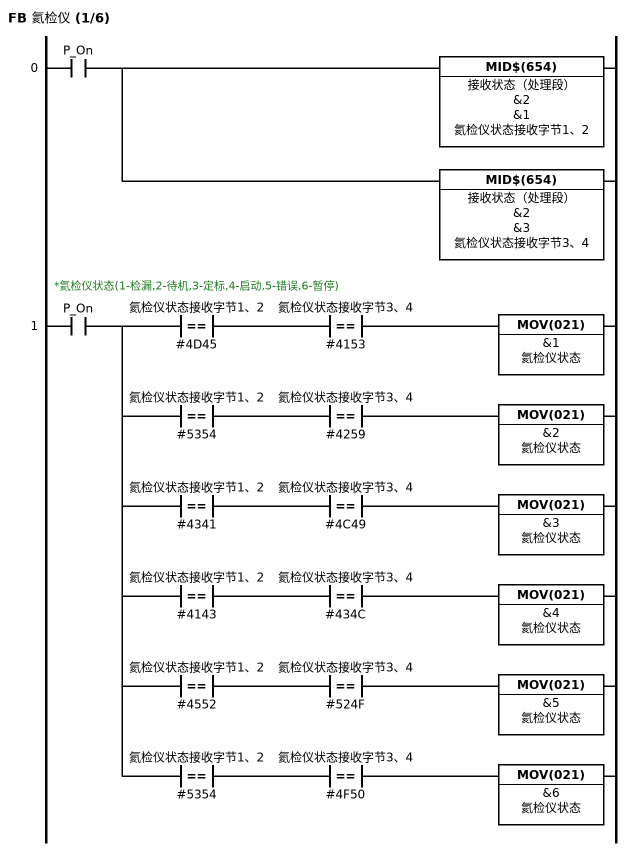
; rung 0
LD P_On
MID$(654) 接收状态（处理段） &2 &1 氦检仪状态接收字节1、2
MID$(654) 接收状态（处理段） &2 &3 氦检仪状态接收字节3、4
; rung 1: *氦检仪状态(1-检漏,2-待机,3-定标,4-启动,5-错误,6-暂停)
LD P_On
OUT TR0
AND=(300) 氦检仪状态接收字节1、2 #4D45
AND=(300) 氦检仪状态接收字节3、4 #4153
MOV(021) &1 氦检仪状态
LD TR0
AND=(300) 氦检仪状态接收字节1、2 #5354
AND=(300) 氦检仪状态接收字节3、4 #4259
MOV(021) &2 氦检仪状态
LD TR0
AND=(300) 氦检仪状态接收字节1、2 #4341
AND=(300) 氦检仪状态接收字节3、4 #4C49
MOV(021) &3 氦检仪状态
LD TR0
AND=(300) 氦检仪状态接收字节1、2 #4143
AND=(300) 氦检仪状态接收字节3、4 #434C
MOV(021) &4 氦检仪状态
LD TR0
AND=(300) 氦检仪状态接收字节1、2 #4552
AND=(300) 氦检仪状态接收字节3、4 #524F
MOV(021) &5 氦检仪状态
LD TR0
AND=(300) 氦检仪状态接收字节1、2 #5354
AND=(300) 氦检仪状态接收字节3、4 #4F50
MOV(021) &6 氦检仪状态

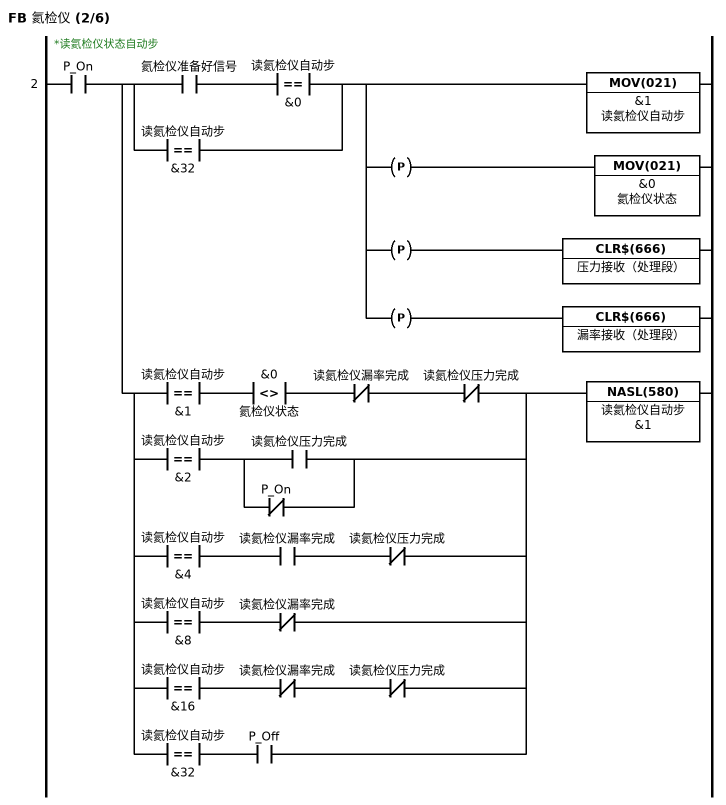
; rung 2: *读氦检仪状态自动步
LD P_On
OUT TR0
LD 氦检仪准备好信号
AND=(300) 读氦检仪自动步 &0
OR=(300) 读氦检仪自动步 &32
ANDLD
OUT TR1
MOV(021) &1 读氦检仪自动步
UP(521)
MOV(021) &0 氦检仪状态
LD TR1
UP(521)
CLR$(666) 压力接收（处理段）
LD TR1
UP(521)
CLR$(666) 漏率接收（处理段）
LD TR0
LD=(300) 读氦检仪自动步 &1
AND<>(305) &0 氦检仪状态
ANDNOT 读氦检仪漏率完成
ANDNOT 读氦检仪压力完成
LD=(300) 读氦检仪自动步 &2
LD 读氦检仪压力完成
ORNOT P_On
ANDLD
ORLD
LD=(300) 读氦检仪自动步 &4
AND 读氦检仪漏率完成
ANDNOT 读氦检仪压力完成
ORLD
LD=(300) 读氦检仪自动步 &8
ANDNOT 读氦检仪漏率完成
ORLD
LD=(300) 读氦检仪自动步 &16
ANDNOT 读氦检仪漏率完成
ANDNOT 读氦检仪压力完成
ORLD
LD=(300) 读氦检仪自动步 &32
AND P_Off
ORLD
ANDLD
NASL(580) 读氦检仪自动步 &1

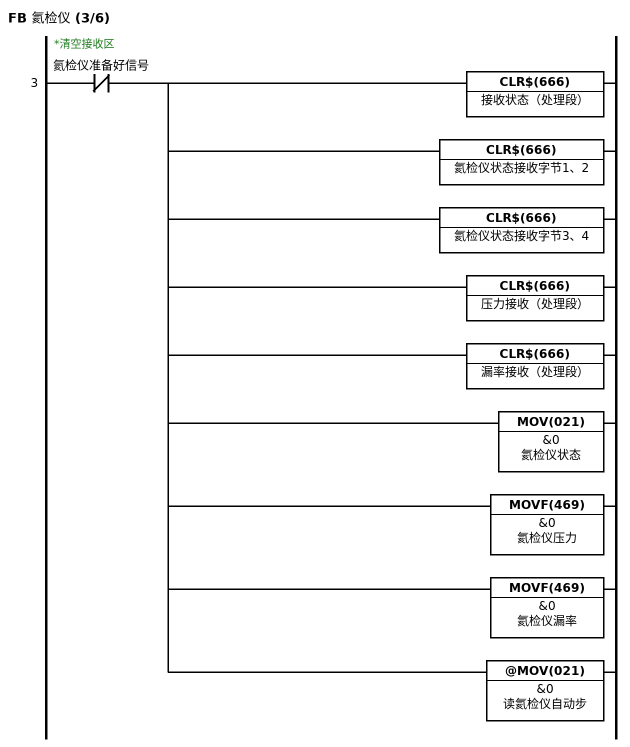
; rung 3: *清空接收区
LDNOT 氦检仪准备好信号
CLR$(666) 接收状态（处理段）
CLR$(666) 氦检仪状态接收字节1、2
CLR$(666) 氦检仪状态接收字节3、4
CLR$(666) 压力接收（处理段）
CLR$(666) 漏率接收（处理段）
MOV(021) &0 氦检仪状态
MOVF(469) &0 氦检仪压力
MOVF(469) &0 氦检仪漏率
@MOV(021) &0 读氦检仪自动步

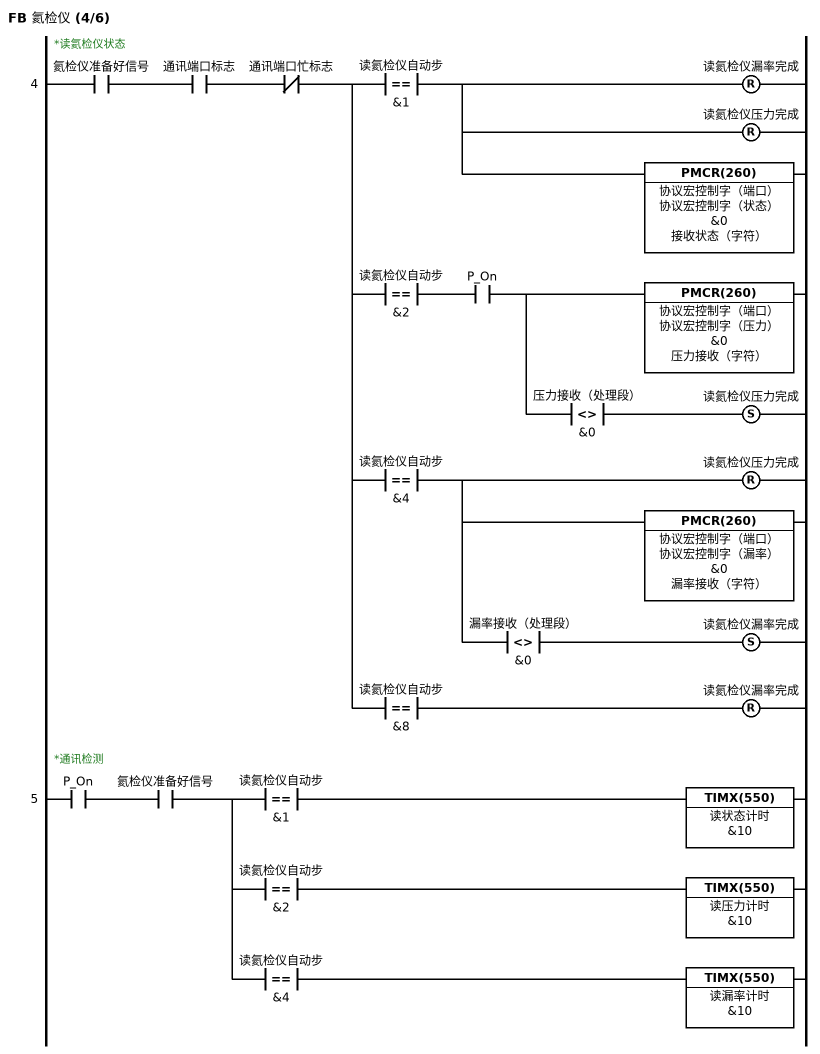
; rung 4: *读氦检仪状态
LD 氦检仪准备好信号
AND 通讯端口标志
ANDNOT 通讯端口忙标志
OUT TR0
AND=(300) 读氦检仪自动步 &1
RSET 读氦检仪漏率完成
RSET 读氦检仪压力完成
PMCR(260) 协议宏控制字（端口） 协议宏控制字（状态） &0 接收状态（字符）
LD TR0
AND=(300) 读氦检仪自动步 &2
AND P_On
PMCR(260) 协议宏控制字（端口） 协议宏控制字（压力） &0 压力接收（字符）
AND<>(305) 压力接收（处理段） &0
SET 读氦检仪压力完成
LD TR0
AND=(300) 读氦检仪自动步 &4
RSET 读氦检仪压力完成
PMCR(260) 协议宏控制字（端口） 协议宏控制字（漏率） &0 漏率接收（字符）
AND<>(305) 漏率接收（处理段） &0
SET 读氦检仪漏率完成
LD TR0
AND=(300) 读氦检仪自动步 &8
RSET 读氦检仪漏率完成
; rung 5: *通讯检测
LD P_On
AND 氦检仪准备好信号
OUT TR0
AND=(300) 读氦检仪自动步 &1
TIMX(550) 读状态计时 &10
LD TR0
AND=(300) 读氦检仪自动步 &2
TIMX(550) 读压力计时 &10
LD TR0
AND=(300) 读氦检仪自动步 &4
TIMX(550) 读漏率计时 &10

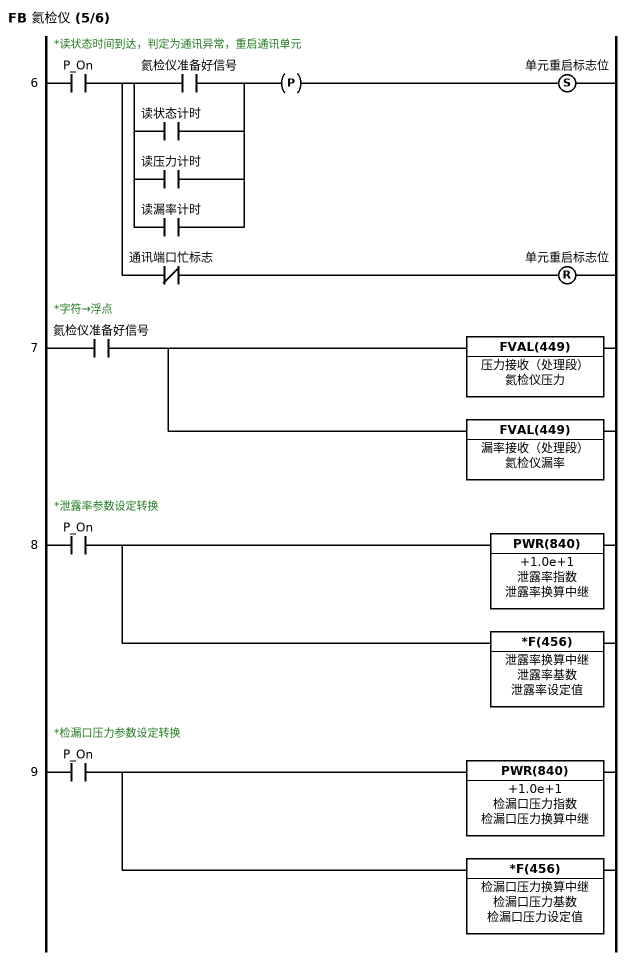
; rung 6: *读状态时间到达，判定为通讯异常，重启通讯单元
LD P_On
OUT TR0
LD 氦检仪准备好信号
OR 读状态计时
OR 读压力计时
OR 读漏率计时
ANDLD
UP(521)
SET 单元重启标志位
LD TR0
ANDNOT 通讯端口忙标志
RSET 单元重启标志位
; rung 7: *字符→浮点
LD 氦检仪准备好信号
FVAL(449) 压力接收（处理段） 氦检仪压力
FVAL(449) 漏率接收（处理段） 氦检仪漏率
; rung 8: *泄露率参数设定转换
LD P_On
PWR(840) +1.0e+1 泄露率指数 泄露率换算中继
*F(456) 泄露率换算中继 泄露率基数 泄露率设定值
; rung 9: *检漏口压力参数设定转换
LD P_On
PWR(840) +1.0e+1 检漏口压力指数 检漏口压力换算中继
*F(456) 检漏口压力换算中继 检漏口压力基数 检漏口压力设定值

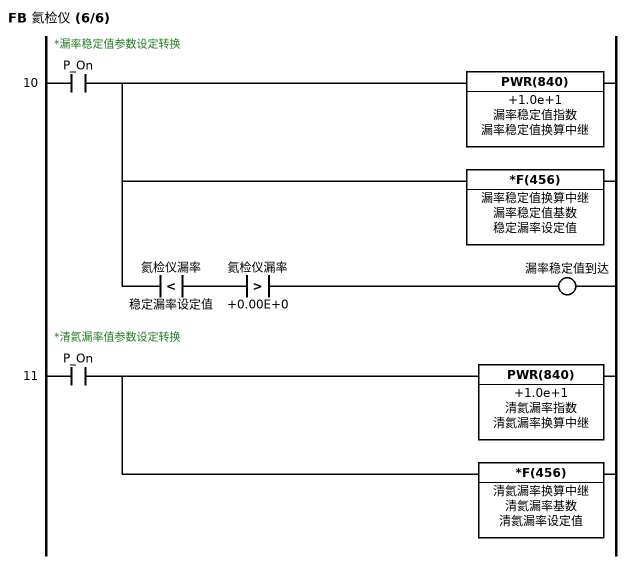
; rung 10: *漏率稳定值参数设定转换
LD P_On
PWR(840) +1.0e+1 漏率稳定值指数 漏率稳定值换算中继
*F(456) 漏率稳定值换算中继 漏率稳定值基数 稳定漏率设定值
AND<F(331) 氦检仪漏率 稳定漏率设定值
AND>F(333) 氦检仪漏率 +0.00E+0
OUT 漏率稳定值到达
; rung 11: *清氦漏率值参数设定转换
LD P_On
PWR(840) +1.0e+1 清氦漏率指数 清氦漏率换算中继
*F(456) 清氦漏率换算中继 清氦漏率基数 清氦漏率设定值

## Function block 腔体自检
VAR_INPUT
  紧急停止 : BOOL;
  真空泵启动信号 : BOOL;
  实时真空值 : REAL;
  自检抽真空设定阀值 : REAL;
  自检破真空设定阀值 : REAL;
  自检抽真空设定时间 : UINT;
  自检保压前设定时间 : UINT;
  自检保压设定时间 : UINT;
  自检泄漏量上限 : REAL;
  腔体顶升气缸上升到位信号 : BOOL;
  腔体顶升气缸下降到位信号 : BOOL;
  平移气缸出料位信号 : BOOL;
  平移气缸氦检位信号 : BOOL;
  抽真空阀状态 : BOOL;
  破真空阀状态 : BOOL;
  抽气阀可打开 : BOOL;
  自检停止（SW） : BOOL;
  自检启动（SW） : BOOL;
  工站初始化 : BOOL;
  腔体在初始位 : BOOL;
END_VAR
VAR_OUTPUT
  功能块运行中 : BOOL;
  自检保压前真空值（PV） : REAL;
  自检保压后真空值（PV） : REAL;
  自检泄漏（PV） : REAL;
  自检结果 : WORD;
  自检开真空泵 : BOOL;
  平移气缸到出料位 : BOOL;
  平移气缸到氦检位 : BOOL;
  自检腔体顶升气缸下降 : BOOL;
  腔体顶升气缸上升 : BOOL;
  自检开抽真空阀 : BOOL;
  自检关抽真空阀 : BOOL;
  自检开破真空阀 : BOOL;
  自检关破真空阀 : BOOL;
  自检保压前实际时间 : WORD;
  自检保压实际时间 : WORD;
  自检抽真空实际时间 : WORD;
  自检完成 : BOOL;
  腔体自检抽真空需求 : BOOL;
  自检保压前真空值2（PV） : REAL;
  自检保压后真空值2（PV） : REAL;
  自检泄漏2（PV） : REAL;
  自检结果2 : WORD;
  自检保压前实际时间2 : WORD;
  自检保压实际时间2 : WORD;
  自检抽真空实际时间2 : WORD;
END_VAR
VAR_IN_OUT
  一号自检 : BOOL;
  二号自检 : BOOL;
END_VAR
VAR
  自检启动 : BOOL;
  自检步序号 : DWORD;
  自检步进条件 : BOOL;
  自检抽真空阀值到达 : BOOL;
  数据运算延时 : TIMER;
  自检破真空阀值到达 : TIMER;
  自检移位 : BOOL;
  自检抽真空定时器 : TIMER;
  自检保压前定时器 : TIMER;
  自检保压定时器 : TIMER;
  自检启动延时 : TIMER;
  自动模式 AT 4.13 : BOOL;  (* 自动模式下禁止功能块运行，直接取I：4.13 *)
END_VAR
; rung 0: *功能块启动,数据初始化
; cells of this rung as drawn
  row 0 col 0: LD P_On
  row 0 col 1: LD 自检停止（SW）
  row 0 col 2: UP(521)
  row 0 col 3: wire
  row 0 col 4: wire
  row 0 col 5: wire
  row 0 col 6: RSET 自检启动
  row 1 col 1: LD 工站初始化
  row 2 col 1: LD 自动模式
  row 2 col 2: wire
  row 2 col 3: wire
  row 2 col 4: wire
  row 2 col 5: wire
  row 2 col 6: RSET 一号自检
  row 3 col 1: LD 紧急停止
  row 3 col 2: wire
  row 4 col 3: wire
  row 4 col 4: wire
  row 4 col 5: wire
  row 4 col 6: RSET 二号自检
  row 6 col 1: LD 自检启动（SW）
  row 6 col 2: UP(521)
  row 6 col 3: LD 腔体在初始位
  row 6 col 4: wire
  row 6 col 5: wire
  row 6 col 6: SET 自检启动
  row 7 col 1: LD 一号自检
  row 8 col 1: LD 二号自检
  row 9 col 1: LD 自检启动
  row 9 col 2: LDNOT 自检启动延时
  row 9 col 3: LDNOT 功能块运行中
  row 9 col 4: LDNOT 二号自检
  row 9 col 5: wire
  row 9 col 6: MOV(021) &0 自检抽真空实际时间
  row 12 col 5: wire
  row 12 col 6: MOV(021) &0 自检保压前实际时间
  row 15 col 5: wire
  row 15 col 6: MOV(021) &0 自检保压实际时间
  row 18 col 5: wire
  row 18 col 6: MOVF(469) &0 自检保压前真空值（PV）
  row 21 col 5: wire
  row 21 col 6: MOVF(469) &0 自检保压后真空值（PV）
  row 24 col 5: wire
  row 24 col 6: MOVF(469) &0 自检泄漏（PV）
  row 27 col 5: wire
  row 27 col 6: MOV(021) &0 自检结果
  row 30 col 4: LDNOT 一号自检
  row 30 col 5: wire
  row 30 col 6: MOV(021) &0 自检抽真空实际时间2
  row 33 col 5: wire
  row 33 col 6: MOV(021) &0 自检保压前实际时间2
  row 36 col 5: wire
  row 36 col 6: MOV(021) &0 自检保压实际时间2
  row 39 col 5: wire
  row 39 col 6: MOVF(469) &0 自检保压前真空值2（PV）
  row 42 col 5: wire
  row 42 col 6: MOVF(469) &0 自检保压后真空值2（PV）
  row 45 col 5: wire
  row 45 col 6: MOVF(469) &0 自检泄漏2（PV）
  row 48 col 5: wire
  row 48 col 6: MOV(021) &0 自检结果2
  vertical links (row, left of col): 0,1 0,2 0,3 1,1 1,3 2,1 2,3 3,1 3,3 4,1 5,1 6,1 6,2 7,1 7,2 8,1 9,4 9,5 10,4 10,5 11,4 11,5 12,4 12,5 13,4 13,5 14,4 14,5 15,4 15,5 16,4 16,5 17,4 17,5 18,4 18,5 19,4 19,5 20,4 20,5 21,4 21,5 22,4 22,5 23,4 23,5 24,4 24,5 25,4 25,5 26,4 26,5 27,4 28,4 29,4 30,5 31,5 32,5 33,5 34,5 35,5 36,5 37,5 38,5 39,5 40,5 41,5 42,5 43,5 44,5 45,5 46,5 47,5

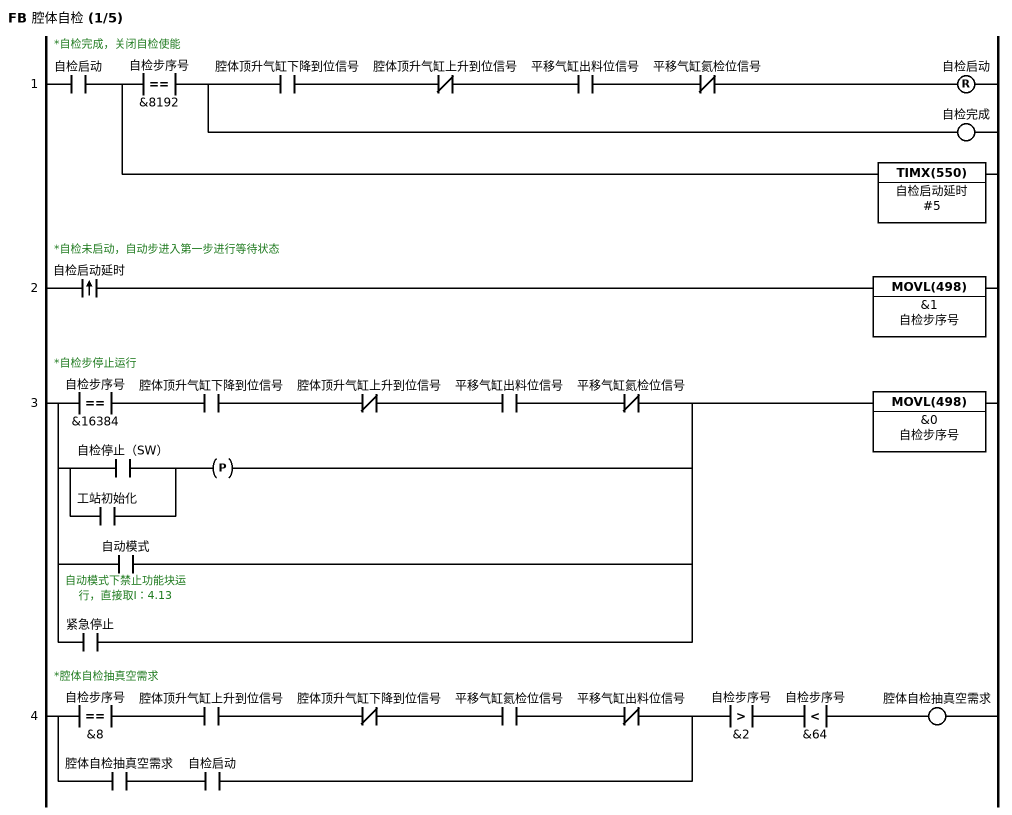
; rung 1: *自检完成，关闭自检使能
LD 自检启动
OUT TR0
AND=(300) 自检步序号 &8192
OUT TR1
AND 腔体顶升气缸下降到位信号
ANDNOT 腔体顶升气缸上升到位信号
AND 平移气缸出料位信号
ANDNOT 平移气缸氦检位信号
RSET 自检启动
LD TR1
OUT 自检完成
LD TR0
TIMX(550) 自检启动延时 #5
; rung 2: *自检未启动，自动步进入第一步进行等待状态
@LD 自检启动延时
MOVL(498) &1 自检步序号
; rung 3: *自检步停止运行
LD=(300) 自检步序号 &16384
AND 腔体顶升气缸下降到位信号
ANDNOT 腔体顶升气缸上升到位信号
AND 平移气缸出料位信号
ANDNOT 平移气缸氦检位信号
LD 自检停止（SW）
OR 工站初始化
UP(521)
ORLD
OR 自动模式  ; 自动模式下禁止功能块运行，直接取I：4.13
OR 紧急停止
MOVL(498) &0 自检步序号
; rung 4: *腔体自检抽真空需求
LD=L(301) 自检步序号 &8
AND 腔体顶升气缸上升到位信号
ANDNOT 腔体顶升气缸下降到位信号
AND 平移气缸氦检位信号
ANDNOT 平移气缸出料位信号
LD 腔体自检抽真空需求
AND 自检启动
ORLD
AND>L(321) 自检步序号 &2
AND<L(311) 自检步序号 &64
OUT 腔体自检抽真空需求

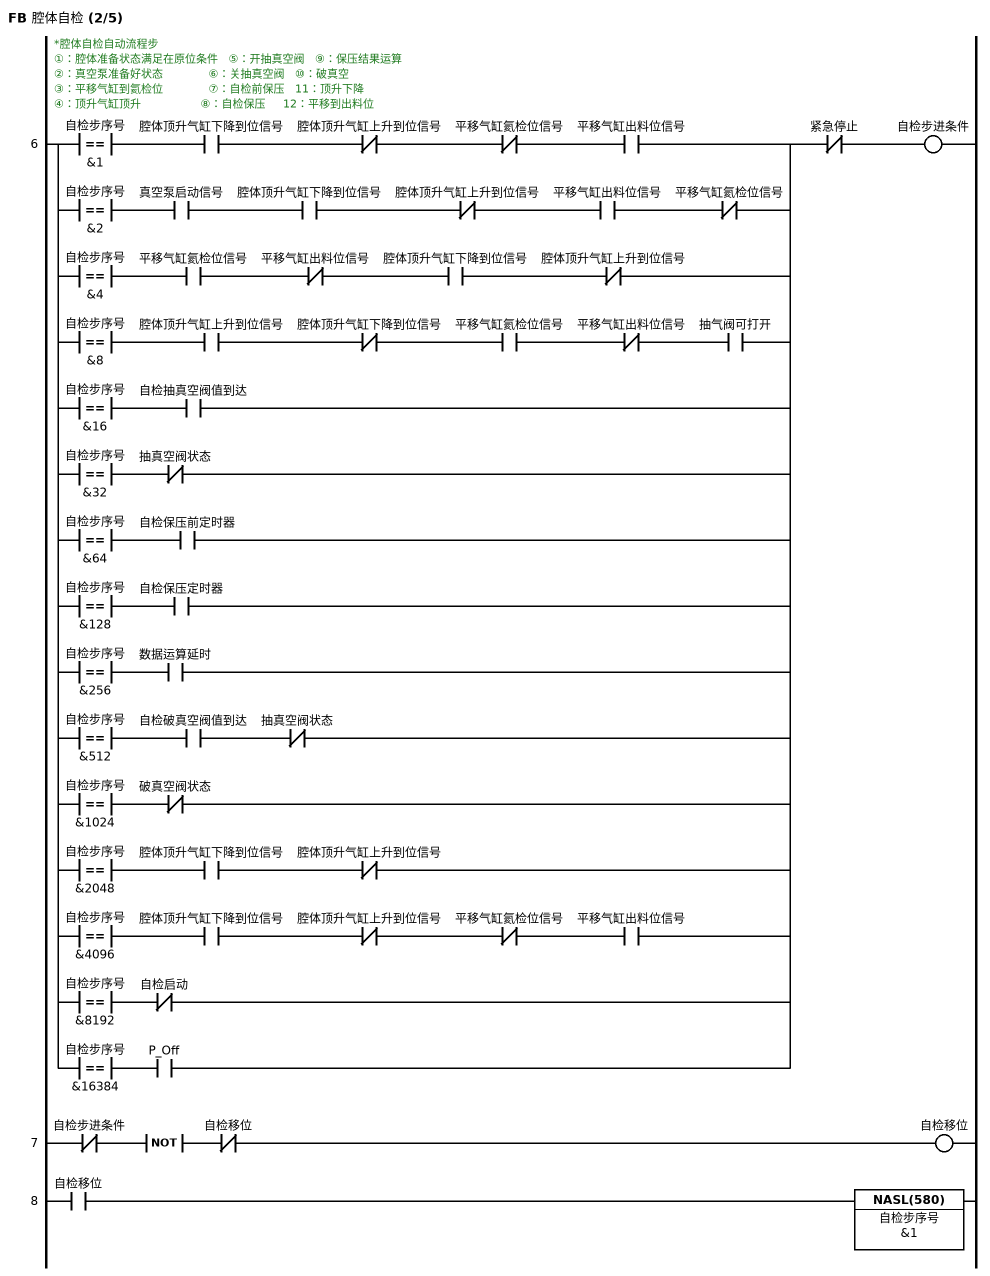
; rung 6: *腔体自检自动流程步 / ①：腔体准备状态满足在原位条件   ⑤：开抽真空阀   ⑨：保压结果运算 / ②：真空泵准备好状态             ⑥：关抽真空阀   ⑩：破真空 / ③：平移气缸到氦检位             ⑦：自检前保压   11：顶升下降 / ④：顶升气缸顶升                 ⑧：自检保压     12：平移到出料位
LD=L(301) 自检步序号 &1
AND 腔体顶升气缸下降到位信号
ANDNOT 腔体顶升气缸上升到位信号
ANDNOT 平移气缸氦检位信号
AND 平移气缸出料位信号
LD=L(301) 自检步序号 &2
AND 真空泵启动信号
AND 腔体顶升气缸下降到位信号
ANDNOT 腔体顶升气缸上升到位信号
AND 平移气缸出料位信号
ANDNOT 平移气缸氦检位信号
ORLD
LD=L(301) 自检步序号 &4
AND 平移气缸氦检位信号
ANDNOT 平移气缸出料位信号
AND 腔体顶升气缸下降到位信号
ANDNOT 腔体顶升气缸上升到位信号
ORLD
LD=L(301) 自检步序号 &8
AND 腔体顶升气缸上升到位信号
ANDNOT 腔体顶升气缸下降到位信号
AND 平移气缸氦检位信号
ANDNOT 平移气缸出料位信号
AND 抽气阀可打开
ORLD
LD=L(301) 自检步序号 &16
AND 自检抽真空阀值到达
ORLD
LD=L(301) 自检步序号 &32
ANDNOT 抽真空阀状态
ORLD
LD=L(301) 自检步序号 &64
AND 自检保压前定时器
ORLD
LD=L(301) 自检步序号 &128
AND 自检保压定时器
ORLD
LD=L(301) 自检步序号 &256
AND 数据运算延时
ORLD
LD=L(301) 自检步序号 &512
AND 自检破真空阀值到达
ANDNOT 抽真空阀状态
ORLD
LD=L(301) 自检步序号 &1024
ANDNOT 破真空阀状态
ORLD
LD=L(301) 自检步序号 &2048
AND 腔体顶升气缸下降到位信号
ANDNOT 腔体顶升气缸上升到位信号
ORLD
LD=L(301) 自检步序号 &4096
AND 腔体顶升气缸下降到位信号
ANDNOT 腔体顶升气缸上升到位信号
ANDNOT 平移气缸氦检位信号
AND 平移气缸出料位信号
ORLD
LD=L(301) 自检步序号 &8192
ANDNOT 自检启动
ORLD
LD=L(301) 自检步序号 &16384
AND P_Off
ORLD
ANDNOT 紧急停止
OUT 自检步进条件
; rung 7
LDNOT 自检步进条件
NOT(520)
ANDNOT 自检移位
OUT 自检移位
; rung 8
LD 自检移位
NASL(580) 自检步序号 &1

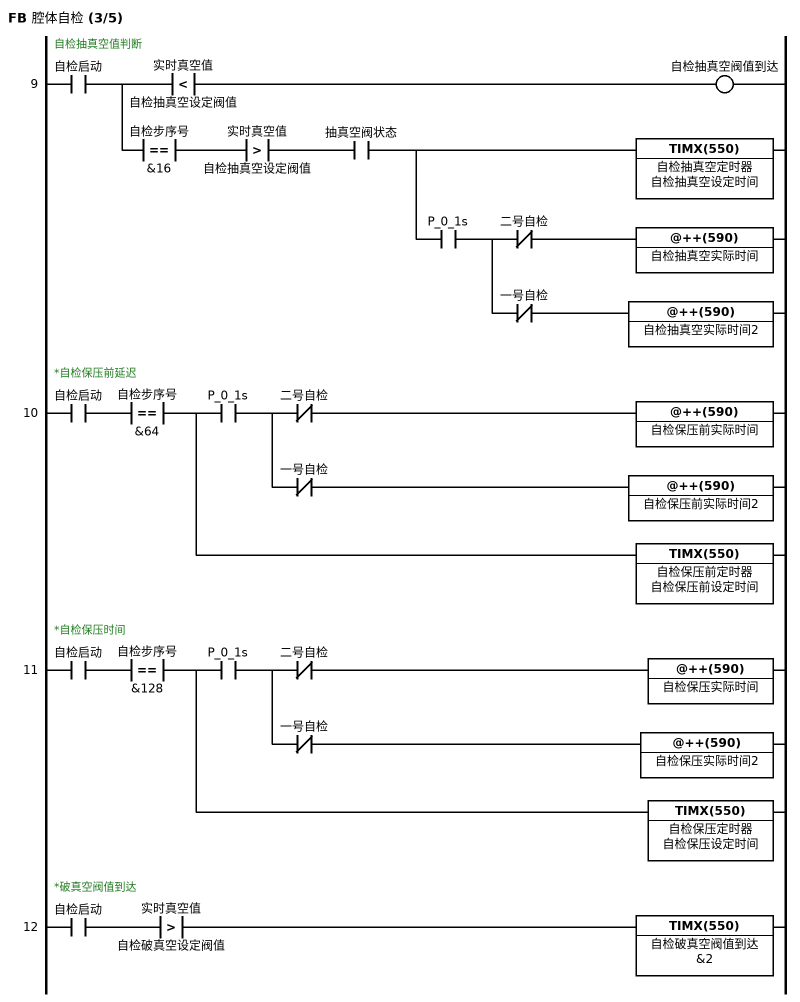
; rung 9: 自检抽真空值判断
LD 自检启动
OUT TR0
AND<F(331) 实时真空值 自检抽真空设定阀值
OUT 自检抽真空阀值到达
LD TR0
AND=L(301) 自检步序号 &16
AND>F(333) 实时真空值 自检抽真空设定阀值
AND 抽真空阀状态
TIMX(550) 自检抽真空定时器 自检抽真空设定时间
AND P_0_1s
OUT TR1
ANDNOT 二号自检
@++(590) 自检抽真空实际时间
LD TR1
ANDNOT 一号自检
@++(590) 自检抽真空实际时间2
; rung 10: *自检保压前延迟
LD 自检启动
AND=L(301) 自检步序号 &64
OUT TR0
AND P_0_1s
OUT TR1
ANDNOT 二号自检
@++(590) 自检保压前实际时间
LD TR1
ANDNOT 一号自检
@++(590) 自检保压前实际时间2
LD TR0
TIMX(550) 自检保压前定时器 自检保压前设定时间
; rung 11: *自检保压时间
LD 自检启动
AND=L(301) 自检步序号 &128
OUT TR0
AND P_0_1s
OUT TR1
ANDNOT 二号自检
@++(590) 自检保压实际时间
LD TR1
ANDNOT 一号自检
@++(590) 自检保压实际时间2
LD TR0
TIMX(550) 自检保压定时器 自检保压设定时间
; rung 12: *破真空阀值到达
LD 自检启动
AND>F(333) 实时真空值 自检破真空设定阀值
TIMX(550) 自检破真空阀值到达 &2

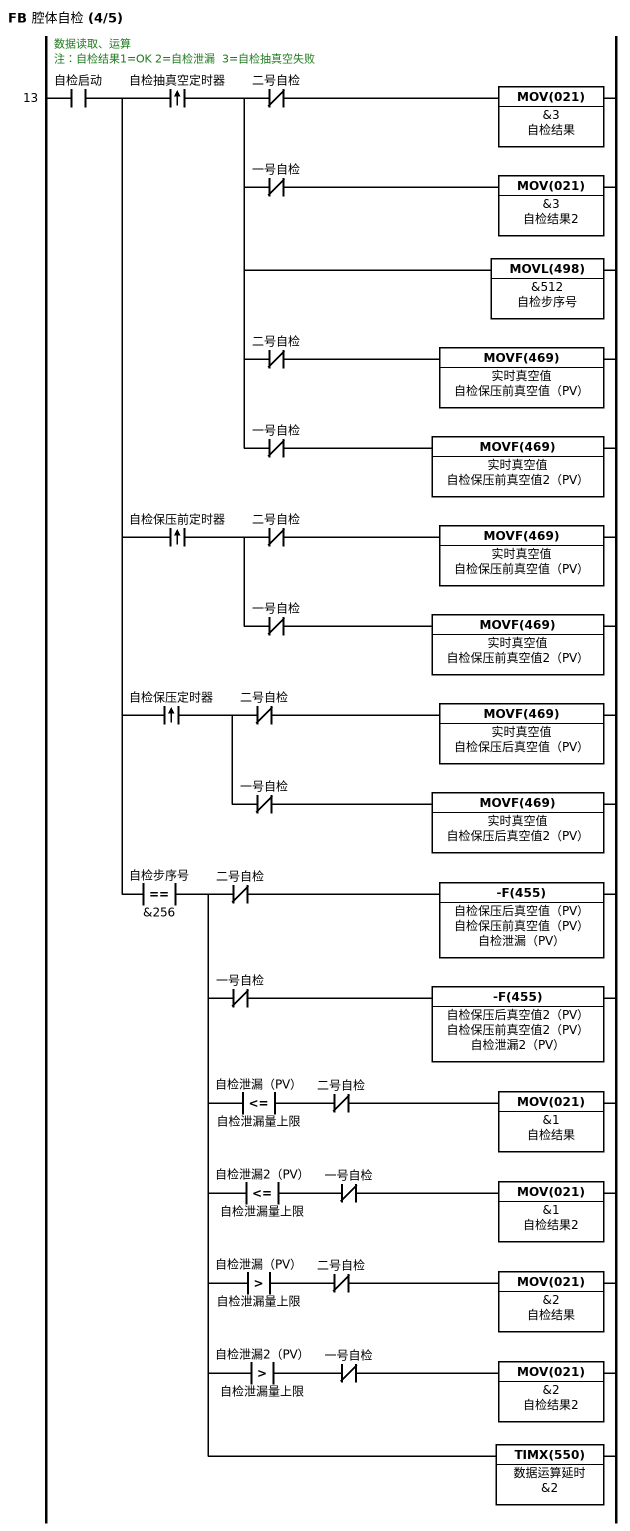
; rung 13: 数据读取、运算 / 注：自检结果1=OK 2=自检泄漏  3=自检抽真空失败
LD 自检启动
OUT TR0
@AND 自检抽真空定时器
OUT TR1
ANDNOT 二号自检
MOV(021) &3 自检结果
LD TR1
ANDNOT 一号自检
MOV(021) &3 自检结果2
LD TR1
MOVL(498) &512 自检步序号
ANDNOT 二号自检
MOVF(469) 实时真空值 自检保压前真空值（PV）
LD TR1
ANDNOT 一号自检
MOVF(469) 实时真空值 自检保压前真空值2（PV）
LD TR0
@AND 自检保压前定时器
OUT TR2
ANDNOT 二号自检
MOVF(469) 实时真空值 自检保压前真空值（PV）
LD TR2
ANDNOT 一号自检
MOVF(469) 实时真空值 自检保压前真空值2（PV）
LD TR0
@AND 自检保压定时器
OUT TR3
ANDNOT 二号自检
MOVF(469) 实时真空值 自检保压后真空值（PV）
LD TR3
ANDNOT 一号自检
MOVF(469) 实时真空值 自检保压后真空值2（PV）
LD TR0
AND=L(301) 自检步序号 &256
OUT TR4
ANDNOT 二号自检
-F(455) 自检保压后真空值（PV） 自检保压前真空值（PV） 自检泄漏（PV）
LD TR4
ANDNOT 一号自检
-F(455) 自检保压后真空值2（PV） 自检保压前真空值2（PV） 自检泄漏2（PV）
LD TR4
AND<=F(332) 自检泄漏（PV） 自检泄漏量上限
ANDNOT 二号自检
MOV(021) &1 自检结果
LD TR4
AND<=F(332) 自检泄漏2（PV） 自检泄漏量上限
ANDNOT 一号自检
MOV(021) &1 自检结果2
LD TR4
AND>F(333) 自检泄漏（PV） 自检泄漏量上限
ANDNOT 二号自检
MOV(021) &2 自检结果
LD TR4
AND>F(333) 自检泄漏2（PV） 自检泄漏量上限
ANDNOT 一号自检
MOV(021) &2 自检结果2
LD TR4
TIMX(550) 数据运算延时 &2

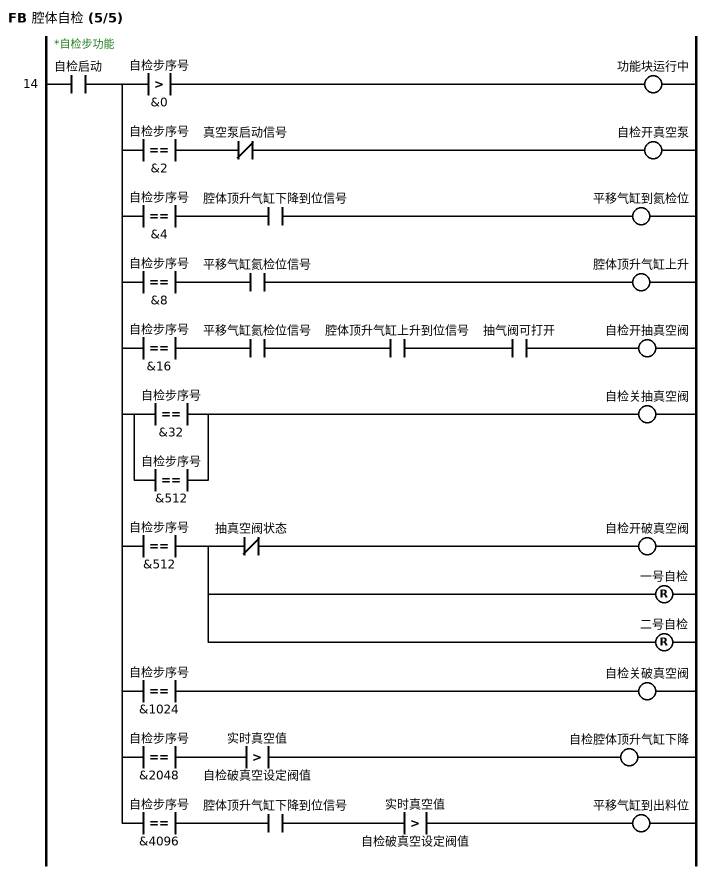
; rung 14: *自检步功能
LD 自检启动
OUT TR0
AND>L(321) 自检步序号 &0
OUT 功能块运行中
LD TR0
AND=L(301) 自检步序号 &2
ANDNOT 真空泵启动信号
OUT 自检开真空泵
LD TR0
AND=L(301) 自检步序号 &4
AND 腔体顶升气缸下降到位信号
OUT 平移气缸到氦检位
LD TR0
AND=L(301) 自检步序号 &8
AND 平移气缸氦检位信号
OUT 腔体顶升气缸上升
LD TR0
AND=L(301) 自检步序号 &16
AND 平移气缸氦检位信号
AND 腔体顶升气缸上升到位信号
AND 抽气阀可打开
OUT 自检开抽真空阀
LD TR0
LD=L(301) 自检步序号 &32
OR=L(301) 自检步序号 &512
ANDLD
OUT 自检关抽真空阀
LD TR0
AND=L(301) 自检步序号 &512
OUT TR1
ANDNOT 抽真空阀状态
OUT 自检开破真空阀
LD TR1
RSET 一号自检
RSET 二号自检
LD TR0
AND=L(301) 自检步序号 &1024
OUT 自检关破真空阀
LD TR0
AND=L(301) 自检步序号 &2048
AND>F(333) 实时真空值 自检破真空设定阀值
OUT 自检腔体顶升气缸下降
LD TR0
AND=L(301) 自检步序号 &4096
AND 腔体顶升气缸下降到位信号
AND>F(333) 实时真空值 自检破真空设定阀值
OUT 平移气缸到出料位

## Function block 真空计
VAR_INPUT
  in_channel : INT;  (* 模拟量输入通道 *)
END_VAR
VAR_OUTPUT
  fout_value : REAL;  (* 真空计输出(浮点) *)
END_VAR
VAR
  ichannel_value : INT;  (* 模拟量储存 *)
  fchannel_value : REAL;  (* 模拟量(浮点) *)
  fchange_value1 : REAL;  (* 真空计转换1(浮点) *)
  fchange_value2 : REAL;  (* 真空计转换2(浮点) *)
  fchange_value3 : REAL;  (* 真空计转换3(浮点) *)
  fchange_value4 : REAL;  (* 真空计转换4(浮点) *)
  ichannel1_value : DINT;
END_VAR

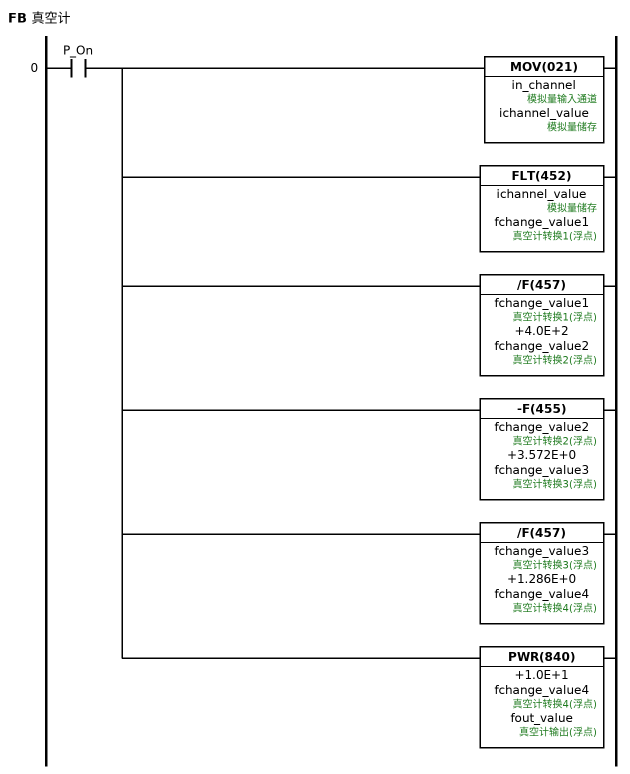
; rung 0
LD P_On
MOV(021) in_channel ichannel_value  ; 模拟量输入通道, 模拟量储存
FLT(452) ichannel_value fchange_value1  ; 模拟量储存, 真空计转换1(浮点)
/F(457) fchange_value1 +4.0E+2 fchange_value2  ; 真空计转换1(浮点), 真空计转换2(浮点)
-F(455) fchange_value2 +3.572E+0 fchange_value3  ; 真空计转换2(浮点), 真空计转换3(浮点)
/F(457) fchange_value3 +1.286E+0 fchange_value4  ; 真空计转换3(浮点), 真空计转换4(浮点)
PWR(840) +1.0E+1 fchange_value4 fout_value  ; 真空计转换4(浮点), 真空计输出(浮点)